// SIMATIC S7-200 SMART project (STEP 7-Micro/WIN SMART), CPU ST40

SYMBOL_TABLE System Symbols
Always_On        SM0.0    // Always ON
RUN_Power_Up     SM0.3    // ON for 1 scan cycle when RUN mode is entered from a power-up condition
END_SYMBOL_TABLE

ORGANIZATION_BLOCK MAIN:OB1
TITLE=Program Comments
BEGIN
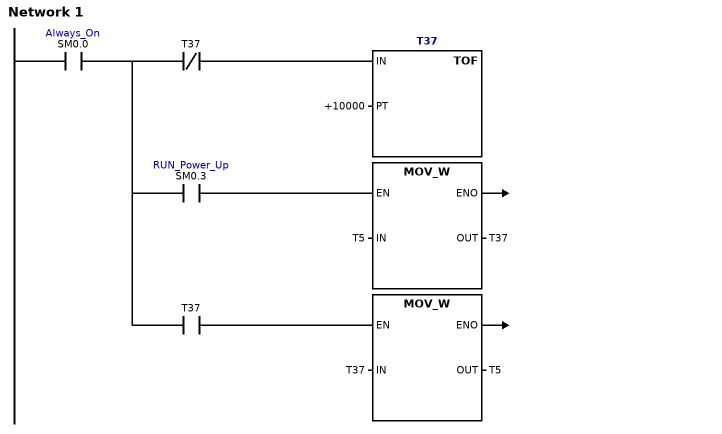
Network 1
LD     Always_On:SM0.0
LPS
AN     T37
TOF    T37, +10000
LRD
A      RUN_Power_Up:SM0.3
MOVW   T5, T37
LPP
A      T37
MOVW   T37, T5
END_ORGANIZATION_BLOCK
